TYPE ST_System_BSp_KueW_Parameter :
STRUCT
	AutoQuittierung					: BOOL	 := 0;

	Stellwert_Temperatur_KW_Max		: REAL	:= 20;
	Stellwert_Temperatur_KW_Min		: REAL	:= 5;
	Stellwert_Temperatur_WW_Max		: REAL	:= 50;
	Stellwert_Temperatur_WW_Min		: REAL	:= 30;
	Kennlinie_Tctr			: DINT := 5000;
END_STRUCT
END_TYPE

(* stored: Version 1.1.0.1, ProductVersion 3.1.4024.9
   DUT ST_System_BSp_KueW_Parameter: Id {42d444b7-9b1f-4500-ac4c-6036d8003b0a} *)
